// TIA Portal V16 export
// export: Created 2024-09-05T17:39:14.3690723Z, ExportSetting WithDefaults, DisplayName Totally Integrated Automation Portal, DisplayVersion V16 Update 6, DisplayName TIA Portal Version Control Interface, DisplayVersion V16 Update 2, DisplayName TIA Portal Openness, DisplayVersion V16 Update 6, DisplayName STEP 7 Professional, DisplayVersion V16 Update 6, DisplayName STEP 7 Safety, DisplayVersion V16, DisplayName WinCC Advanced, DisplayVersion V16 Update 6
FUNCTION "FC_ByteToCharacters" : Void   // FC1071, LAD
{ S7_Optimized_Access := 'FALSE' }
VERSION : 0.1
// stored: AutoNumber false, IsIECCheckEnabled false, SetENOAutomatically false, UDAEnableTagReadback false
   VAR_INPUT
      iByte : Byte;
   END_VAR
   VAR_OUTPUT
      qChar1 : Char;
      qChar2 : Char;
   END_VAR
   VAR_TEMP
      "b" : Byte;
      char1_value : UInt;
      char2_value : UInt;
   END_VAR
   VAR_TEMP   // added for the SCL form of the ladder/FBD networks
      _w1 : Bool;
      _w2 : Bool;
   END_VAR
BEGIN

REGION Network 1: Load input byte to temporary
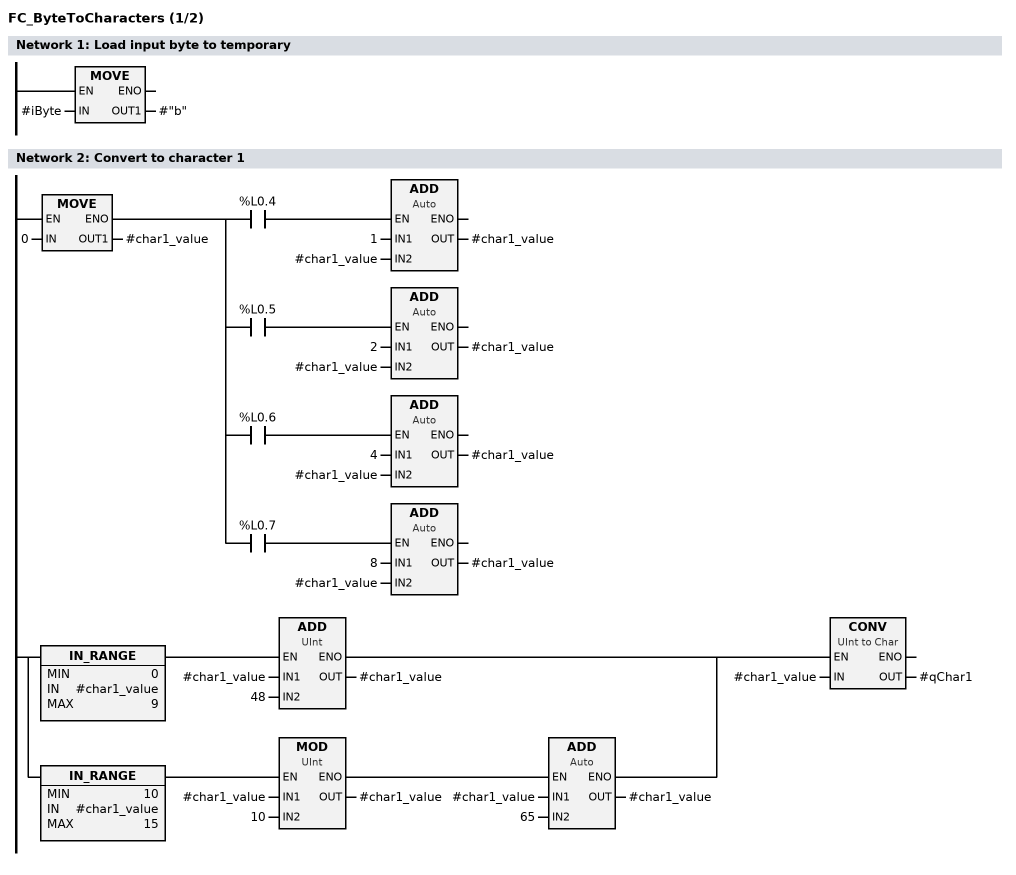
   RUNG wire#powerrail
      Move(in := #iByte, out1 => #"b")
   END_RUNG
   // the same network as SCL:
   #"b" := #iByte;
END_REGION

REGION Network 2: Convert to character 1
   RUNG wire#powerrail
      Move(in := 0, out1 => #char1_value)
      wire#w1
      Contact( %L0.4 )
      Add(in1 := 1, in2 := #char1_value, out => #char1_value)
   END_RUNG
   RUNG wire#w1
      Contact( %L0.5 )
      Add(in1 := 2, in2 := #char1_value, out => #char1_value)
   END_RUNG
   RUNG wire#w1
      Contact( %L0.6 )
      Add(in1 := 4, in2 := #char1_value, out => #char1_value)
   END_RUNG
   RUNG wire#w1
      Contact( %L0.7 )
      Add(in1 := 8, in2 := #char1_value, out => #char1_value)
   END_RUNG
   RUNG wire#powerrail
      { S7_Templates := "SrcType := UInt" } InRange(min := 0, in := #char1_value, max := 9)
      { S7_Templates := "SrcType := UInt" } Add(in1 := #char1_value, in2 := 48, out => #char1_value)
      wire#w2
      { S7_Templates := "[SrcType := UInt, DestType := Char]" } Convert(in := #char1_value, out => #qChar1)
   END_RUNG
   RUNG wire#powerrail
      { S7_Templates := "SrcType := UInt" } InRange(min := 10, in := #char1_value, max := 15)
      { S7_Templates := "SrcType := UInt" } Mod(in1 := #char1_value, in2 := 10, out => #char1_value)
      Add(in1 := #char1_value, in2 := 65, out => #char1_value)
   END_RUNG wire#w2
   // the same network as SCL:
   #char1_value := 0;
   IF %L0.4 THEN #char1_value := 1 + #char1_value; END_IF;
   IF %L0.5 THEN #char1_value := 2 + #char1_value; END_IF;
   IF %L0.6 THEN #char1_value := 4 + #char1_value; END_IF;
   IF %L0.7 THEN #char1_value := 8 + #char1_value; END_IF;
   #_w1 := (0 <= #char1_value) AND (#char1_value <= 9);
   IF #_w1 THEN #char1_value := #char1_value + 48; END_IF;
   #_w2 := (10 <= #char1_value) AND (#char1_value <= 15);
   IF #_w2 THEN
       #char1_value := #char1_value MOD 10;
       #char1_value := #char1_value + 65;
   END_IF;
   IF #_w1 OR #_w2 THEN #qChar1 := UINT_TO_CHAR(#char1_value); END_IF;
END_REGION

REGION Network 3: Convert to character 2
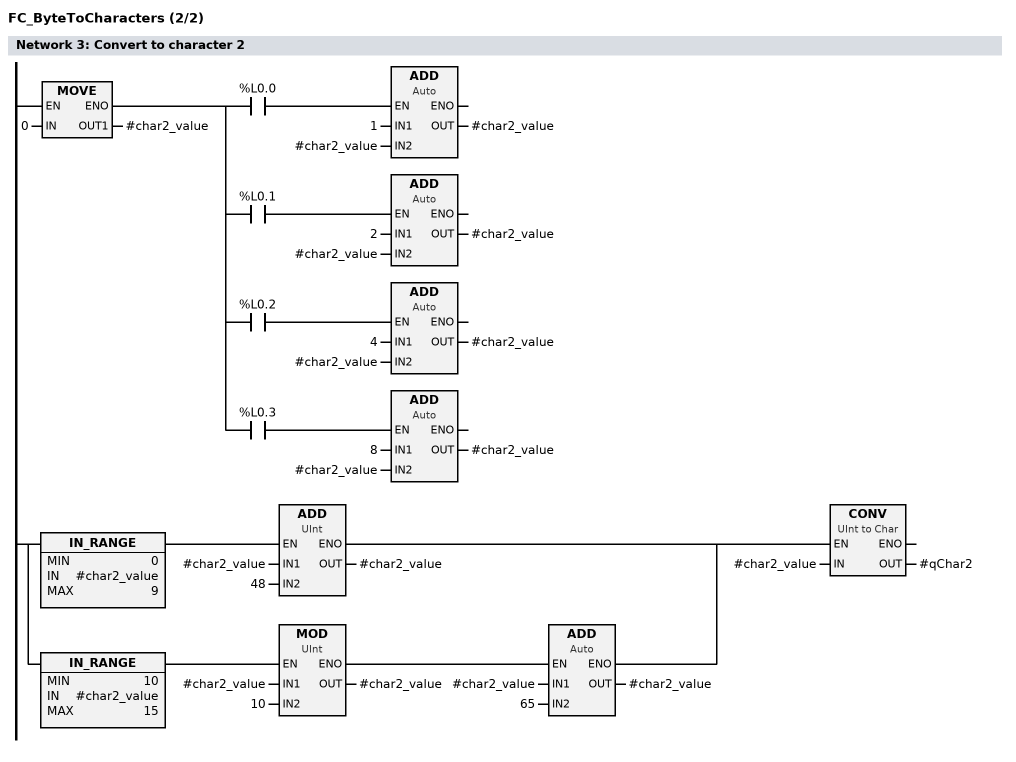
   RUNG wire#powerrail
      Move(in := 0, out1 => #char2_value)
      wire#w1
      Contact( %L0.0 )
      Add(in1 := 1, in2 := #char2_value, out => #char2_value)
   END_RUNG
   RUNG wire#w1
      Contact( %L0.1 )
      Add(in1 := 2, in2 := #char2_value, out => #char2_value)
   END_RUNG
   RUNG wire#w1
      Contact( %L0.2 )
      Add(in1 := 4, in2 := #char2_value, out => #char2_value)
   END_RUNG
   RUNG wire#w1
      Contact( %L0.3 )
      Add(in1 := 8, in2 := #char2_value, out => #char2_value)
   END_RUNG
   RUNG wire#powerrail
      { S7_Templates := "SrcType := UInt" } InRange(min := 0, in := #char2_value, max := 9)
      { S7_Templates := "SrcType := UInt" } Add(in1 := #char2_value, in2 := 48, out => #char2_value)
      wire#w2
      { S7_Templates := "[SrcType := UInt, DestType := Char]" } Convert(in := #char2_value, out => #qChar2)
   END_RUNG
   RUNG wire#powerrail
      { S7_Templates := "SrcType := UInt" } InRange(min := 10, in := #char2_value, max := 15)
      { S7_Templates := "SrcType := UInt" } Mod(in1 := #char2_value, in2 := 10, out => #char2_value)
      Add(in1 := #char2_value, in2 := 65, out => #char2_value)
   END_RUNG wire#w2
   // the same network as SCL:
   #char2_value := 0;
   IF %L0.0 THEN #char2_value := 1 + #char2_value; END_IF;
   IF %L0.1 THEN #char2_value := 2 + #char2_value; END_IF;
   IF %L0.2 THEN #char2_value := 4 + #char2_value; END_IF;
   IF %L0.3 THEN #char2_value := 8 + #char2_value; END_IF;
   #_w1 := (0 <= #char2_value) AND (#char2_value <= 9);
   IF #_w1 THEN #char2_value := #char2_value + 48; END_IF;
   #_w2 := (10 <= #char2_value) AND (#char2_value <= 15);
   IF #_w2 THEN
       #char2_value := #char2_value MOD 10;
       #char2_value := #char2_value + 65;
   END_IF;
   IF #_w1 OR #_w2 THEN #qChar2 := UINT_TO_CHAR(#char2_value); END_IF;
END_REGION
END_FUNCTION
